FUNCTION_BLOCK FB_Syntax_StringLiterals
VAR
    sA  : STRING(255);
    sB  : STRING(255);
    wsC : WSTRING(128);
    sD  : STRING(255);
    sE  : STRING(255);
END_VAR

sA  := 'part1 $' part2';
sB  := 'price $$100';
wsC := "wide string literal";
sD  := 'ae oe ue';
sE  := CONCAT('abc', 'def');

END_FUNCTION_BLOCK

(* stored: Version 1.1.0.1, ProductVersion 3.1.4024.16
   POU FB_Syntax_StringLiterals: Id {7f7e0906-1c46-418f-975c-e13d57e4a30a}, SpecialFunc None *)
